(* Logix 5000 project; controller Sucrose_Main Emulate 5570 rev 20.12; software revision 20.01; part 13 of 30 *)
(* tags used below, declared in another part *)
   AI_E21_0 : REAL[8];   // Analog Input EN2T_FLX 192.168.1.21
   AI_E21_1 : REAL[8];   // Analog Input EN2T_FLX 192.168.1.21
   AI_E21_2 : REAL[8];   // Analog Input EN2T_FLX 192.168.1.21
   Rung_Comment : BOOL;
   SucroseCIP_RINGMAIN_REMOTE : CIP_REMOTE;
   SucroseFiltration : Area_Program;
(* FiltrationArea_AutoLogic, continued *)

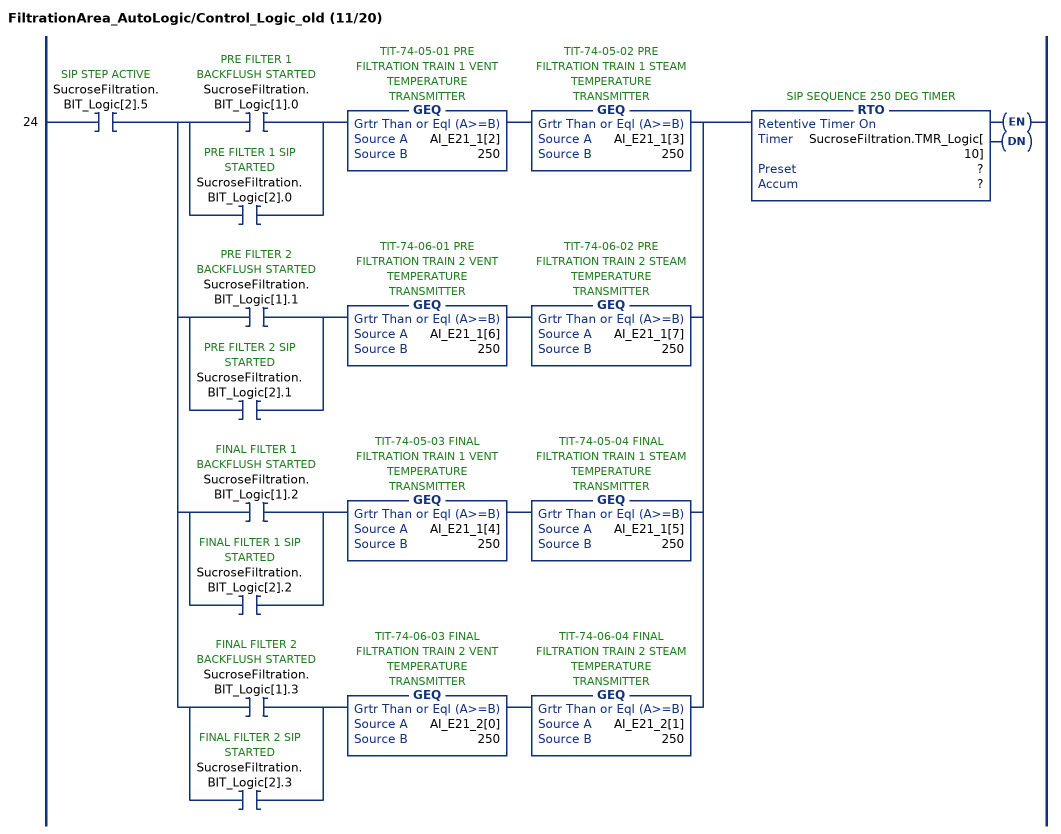
   [picture p232: FiltrationArea_AutoLogic/Control_Logic_old rungs 24-24]
   24: XIC(SucroseFiltration.BIT_Logic[2].5)[[XIC(SucroseFiltration.BIT_Logic[1].0) ,XIC(SucroseFiltration.BIT_Logic[2].0) ] GEQ(AI_E21_1[2],250) GEQ(AI_E21_1[3],250) ,[XIC(SucroseFiltration.BIT_Logic[1].1) ,XIC(SucroseFiltration.BIT_Logic[2].1) ] GEQ(AI_E21_1[6],250) GEQ(AI_E21_1[7],250) ,[XIC(SucroseFiltration.BIT_Logic[1].2) ,XIC(SucroseFiltration.BIT_Logic[2].2) ] GEQ(AI_E21_1[4],250) GEQ(AI_E21_1[5],250) ,[XIC(SucroseFiltration.BIT_Logic[1].3) ,XIC(SucroseFiltration.BIT_Logic[2].3) ] GEQ(AI_E21_2[0],250) GEQ(AI_E21_2[1],250) ]RTO(SucroseFiltration.TMR_Logic[10],?,?);
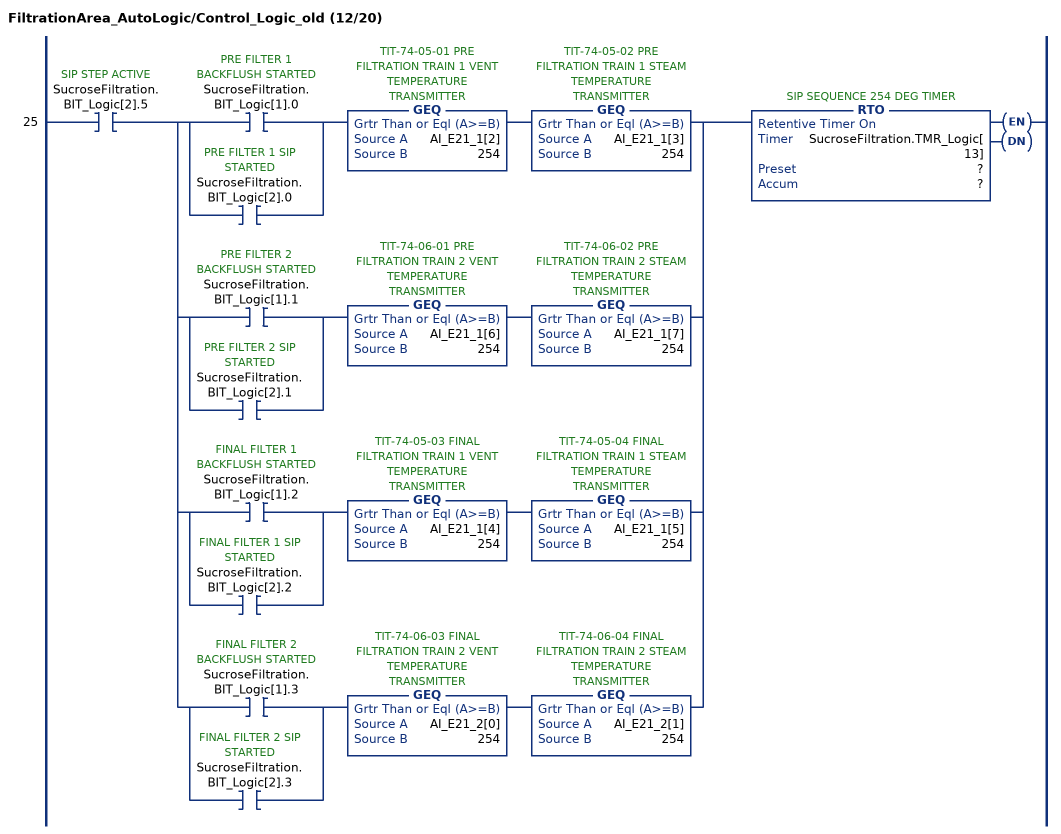
   25: XIC(SucroseFiltration.BIT_Logic[2].5)[[XIC(SucroseFiltration.BIT_Logic[1].0) ,XIC(SucroseFiltration.BIT_Logic[2].0) ] GEQ(AI_E21_1[2],254) GEQ(AI_E21_1[3],254) ,[XIC(SucroseFiltration.BIT_Logic[1].1) ,XIC(SucroseFiltration.BIT_Logic[2].1) ] GEQ(AI_E21_1[6],254) GEQ(AI_E21_1[7],254) ,[XIC(SucroseFiltration.BIT_Logic[1].2) ,XIC(SucroseFiltration.BIT_Logic[2].2) ] GEQ(AI_E21_1[4],254) GEQ(AI_E21_1[5],254) ,[XIC(SucroseFiltration.BIT_Logic[1].3) ,XIC(SucroseFiltration.BIT_Logic[2].3) ] GEQ(AI_E21_2[0],254) GEQ(AI_E21_2[1],254) ]RTO(SucroseFiltration.TMR_Logic[13],?,?);
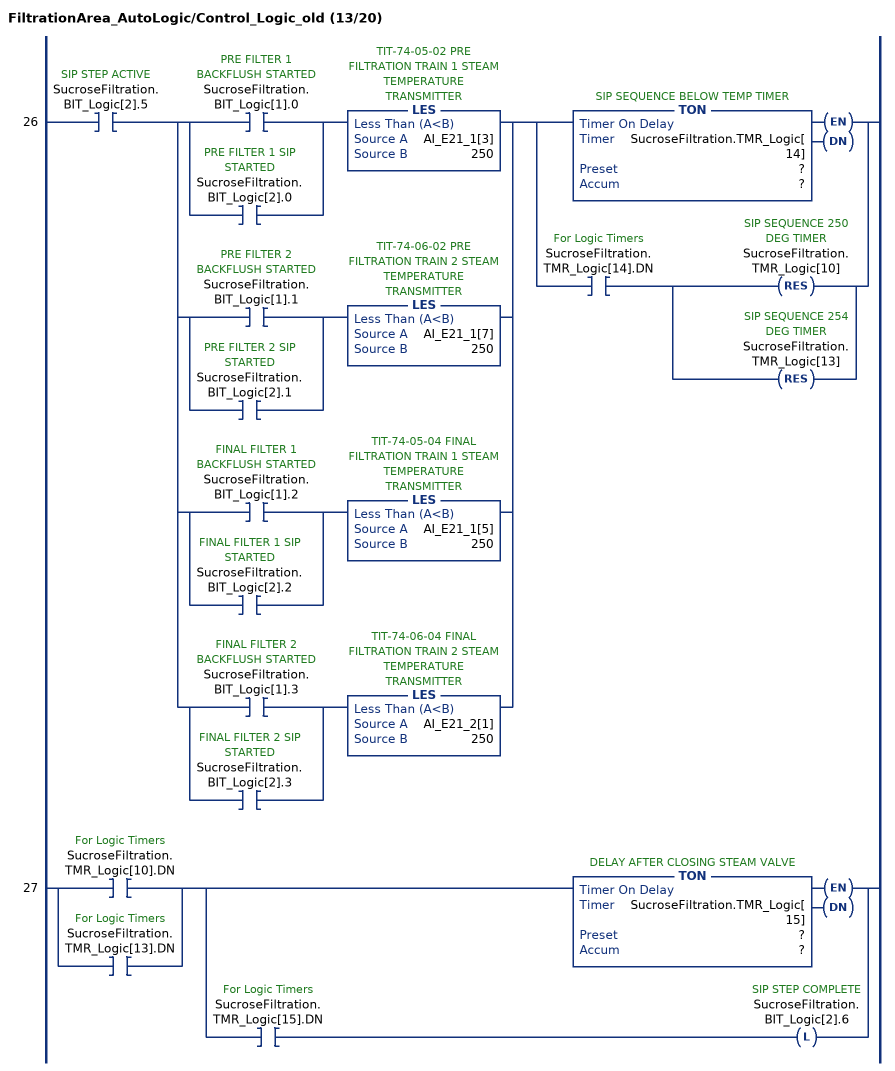
   26: XIC(SucroseFiltration.BIT_Logic[2].5)[[XIC(SucroseFiltration.BIT_Logic[1].0) ,XIC(SucroseFiltration.BIT_Logic[2].0) ] LES(AI_E21_1[3],250) ,[XIC(SucroseFiltration.BIT_Logic[1].1) ,XIC(SucroseFiltration.BIT_Logic[2].1) ] LES(AI_E21_1[7],250) ,[XIC(SucroseFiltration.BIT_Logic[1].2) ,XIC(SucroseFiltration.BIT_Logic[2].2) ] LES(AI_E21_1[5],250) ,[XIC(SucroseFiltration.BIT_Logic[1].3) ,XIC(SucroseFiltration.BIT_Logic[2].3) ] LES(AI_E21_2[1],250) ][TON(SucroseFiltration.TMR_Logic[14],?,?) ,XIC(SucroseFiltration.TMR_Logic[14].DN) [RES(SucroseFiltration.TMR_Logic[10]) ,RES(SucroseFiltration.TMR_Logic[13]) ] ];
   27: [XIC(SucroseFiltration.TMR_Logic[10].DN) ,XIC(SucroseFiltration.TMR_Logic[13].DN) ][TON(SucroseFiltration.TMR_Logic[15],?,?) ,XIC(SucroseFiltration.TMR_Logic[15].DN) OTL(SucroseFiltration.BIT_Logic[2].6) ];
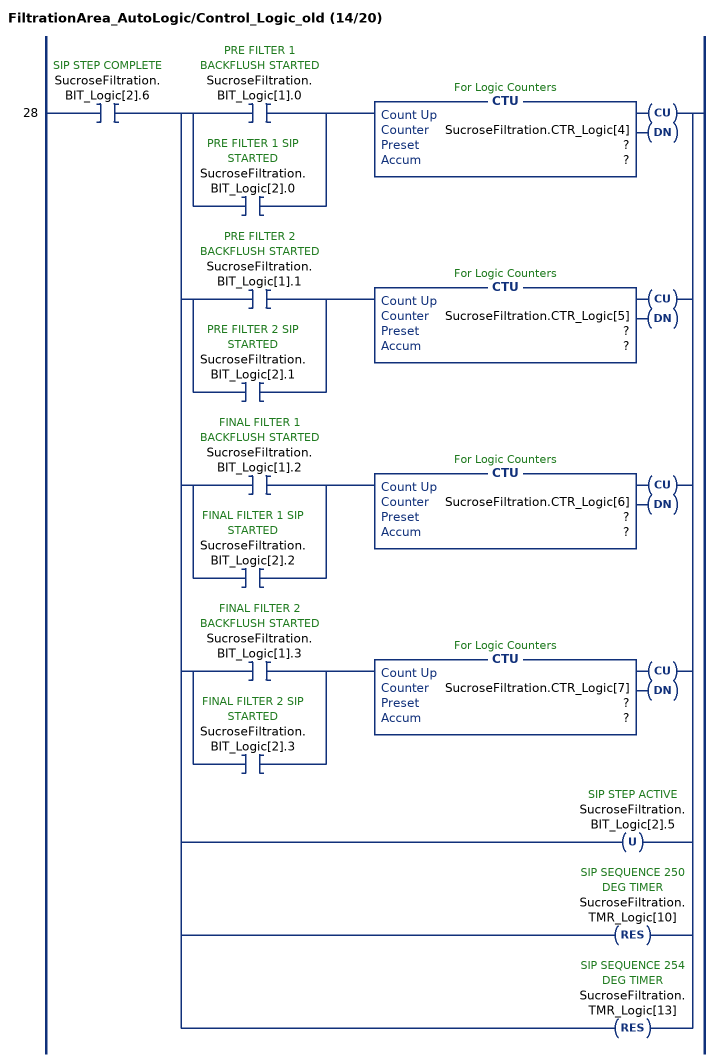
   28: XIC(SucroseFiltration.BIT_Logic[2].6)[[XIC(SucroseFiltration.BIT_Logic[1].0) ,XIC(SucroseFiltration.BIT_Logic[2].0) ] CTU(SucroseFiltration.CTR_Logic[4],?,?) ,[XIC(SucroseFiltration.BIT_Logic[1].1) ,XIC(SucroseFiltration.BIT_Logic[2].1) ] CTU(SucroseFiltration.CTR_Logic[5],?,?) ,[XIC(SucroseFiltration.BIT_Logic[1].2) ,XIC(SucroseFiltration.BIT_Logic[2].2) ] CTU(SucroseFiltration.CTR_Logic[6],?,?) ,[XIC(SucroseFiltration.BIT_Logic[1].3) ,XIC(SucroseFiltration.BIT_Logic[2].3) ] CTU(SucroseFiltration.CTR_Logic[7],?,?) ,OTU(SucroseFiltration.BIT_Logic[2].5) ,RES(SucroseFiltration.TMR_Logic[10]) ,RES(SucroseFiltration.TMR_Logic[13]) ];
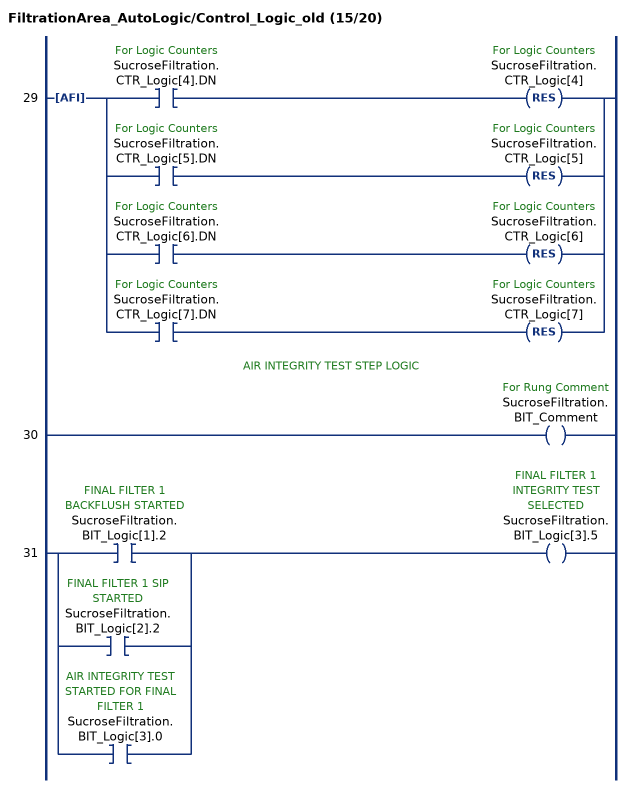
   29: AFI()[XIC(SucroseFiltration.CTR_Logic[4].DN) RES(SucroseFiltration.CTR_Logic[4]) ,XIC(SucroseFiltration.CTR_Logic[5].DN) RES(SucroseFiltration.CTR_Logic[5]) ,XIC(SucroseFiltration.CTR_Logic[6].DN) RES(SucroseFiltration.CTR_Logic[6]) ,XIC(SucroseFiltration.CTR_Logic[7].DN) RES(SucroseFiltration.CTR_Logic[7]) ];
   // AIR INTEGRITY TEST STEP LOGIC
   30: OTE(SucroseFiltration.BIT_Comment);
   31: [XIC(SucroseFiltration.BIT_Logic[1].2) ,XIC(SucroseFiltration.BIT_Logic[2].2) ,XIC(SucroseFiltration.BIT_Logic[3].0) ]OTE(SucroseFiltration.BIT_Logic[3].5);
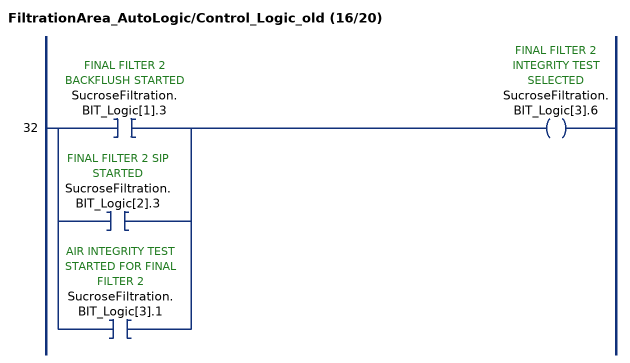
   32: [XIC(SucroseFiltration.BIT_Logic[1].3) ,XIC(SucroseFiltration.BIT_Logic[2].3) ,XIC(SucroseFiltration.BIT_Logic[3].1) ]OTE(SucroseFiltration.BIT_Logic[3].6);
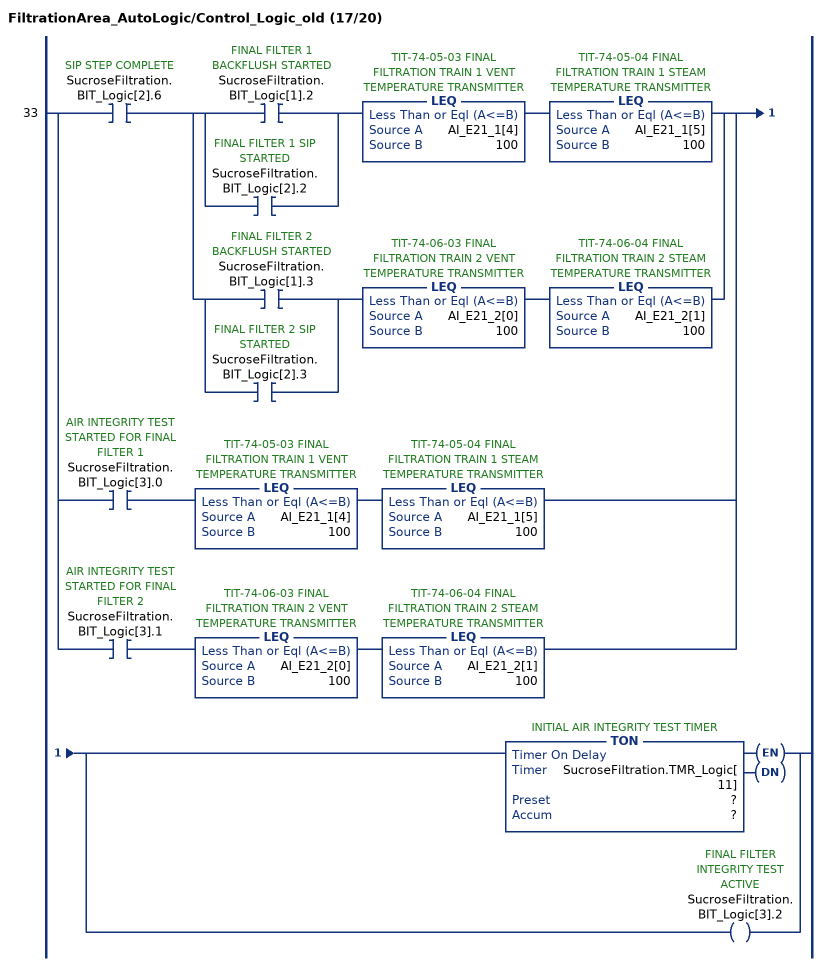
   33: [XIC(SucroseFiltration.BIT_Logic[2].6) [[XIC(SucroseFiltration.BIT_Logic[1].2) ,XIC(SucroseFiltration.BIT_Logic[2].2) ] LEQ(AI_E21_1[4],100) LEQ(AI_E21_1[5],100) ,[XIC(SucroseFiltration.BIT_Logic[1].3) ,XIC(SucroseFiltration.BIT_Logic[2].3) ] LEQ(AI_E21_2[0],100) LEQ(AI_E21_2[1],100) ] ,[XIC(SucroseFiltration.BIT_Logic[3].0) LEQ(AI_E21_1[4],100) LEQ(AI_E21_1[5],100) ,XIC(SucroseFiltration.BIT_Logic[3].1) LEQ(AI_E21_2[0],100) LEQ(AI_E21_2[1],100) ] ][TON(SucroseFiltration.TMR_Logic[11],?,?) ,OTE(SucroseFiltration.BIT_Logic[3].2) ];
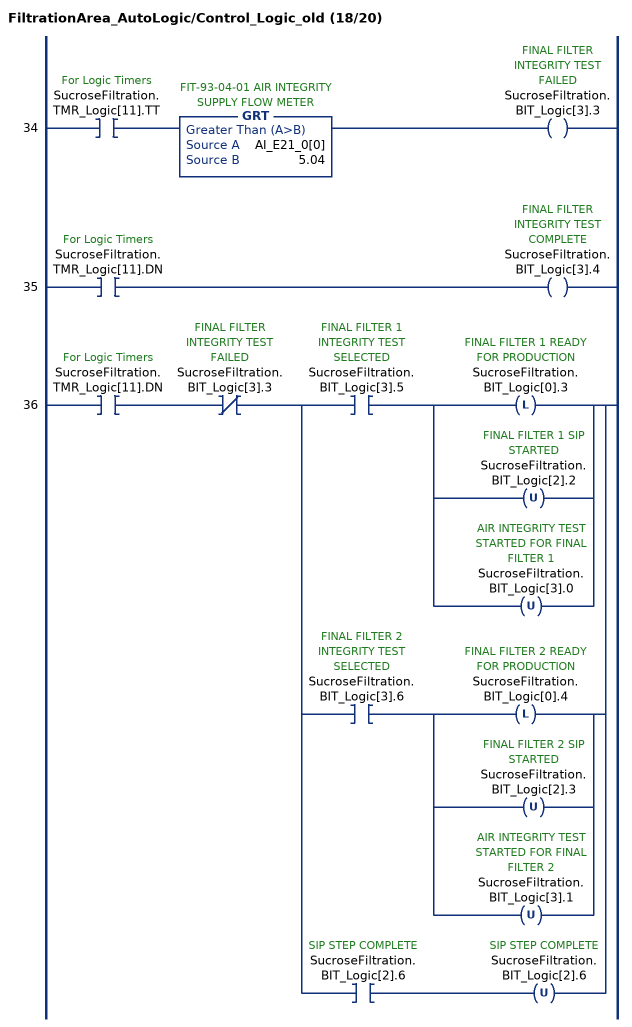
   34: XIC(SucroseFiltration.TMR_Logic[11].TT)GRT(AI_E21_0[0],5.04)OTE(SucroseFiltration.BIT_Logic[3].3);
   35: XIC(SucroseFiltration.TMR_Logic[11].DN)OTE(SucroseFiltration.BIT_Logic[3].4);
   36: XIC(SucroseFiltration.TMR_Logic[11].DN)XIO(SucroseFiltration.BIT_Logic[3].3)[XIC(SucroseFiltration.BIT_Logic[3].5) [OTL(SucroseFiltration.BIT_Logic[0].3) ,OTU(SucroseFiltration.BIT_Logic[2].2) ,OTU(SucroseFiltration.BIT_Logic[3].0) ] ,XIC(SucroseFiltration.BIT_Logic[3].6) [OTL(SucroseFiltration.BIT_Logic[0].4) ,OTU(SucroseFiltration.BIT_Logic[2].3) ,OTU(SucroseFiltration.BIT_Logic[3].1) ] ,XIC(SucroseFiltration.BIT_Logic[2].6) OTU(SucroseFiltration.BIT_Logic[2].6) ];
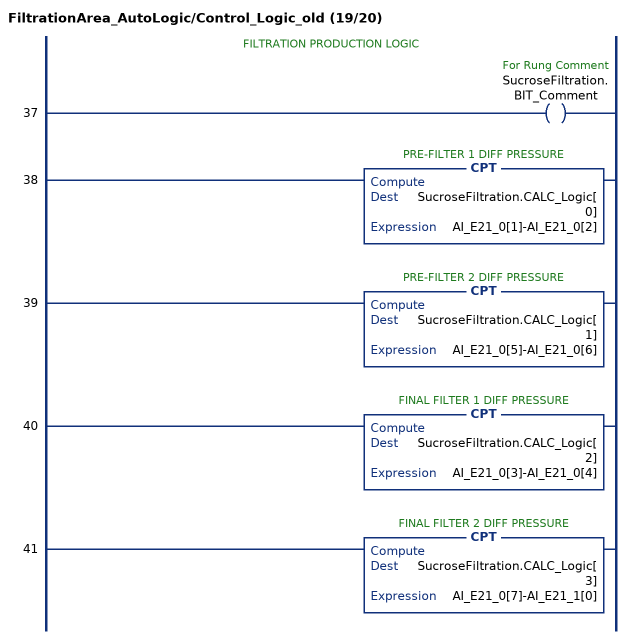
   // FILTRATION PRODUCTION LOGIC
   37: OTE(SucroseFiltration.BIT_Comment);
   38: CPT(SucroseFiltration.CALC_Logic[0],AI_E21_0[1]-AI_E21_0[2]);
   39: CPT(SucroseFiltration.CALC_Logic[1],AI_E21_0[5]-AI_E21_0[6]);
   40: CPT(SucroseFiltration.CALC_Logic[2],AI_E21_0[3]-AI_E21_0[4]);
   41: CPT(SucroseFiltration.CALC_Logic[3],AI_E21_0[7]-AI_E21_1[0]);
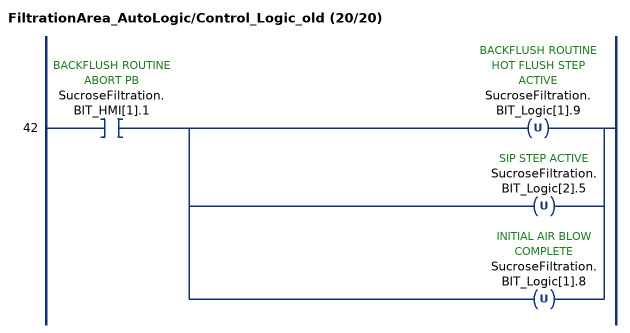
   42: XIC(SucroseFiltration.BIT_HMI[1].1)[OTU(SucroseFiltration.BIT_Logic[1].9) ,OTU(SucroseFiltration.BIT_Logic[2].5) ,OTU(SucroseFiltration.BIT_Logic[1].8) ];
END_ROUTINE

ROUTINE Enable_Logic   (* ladder *)
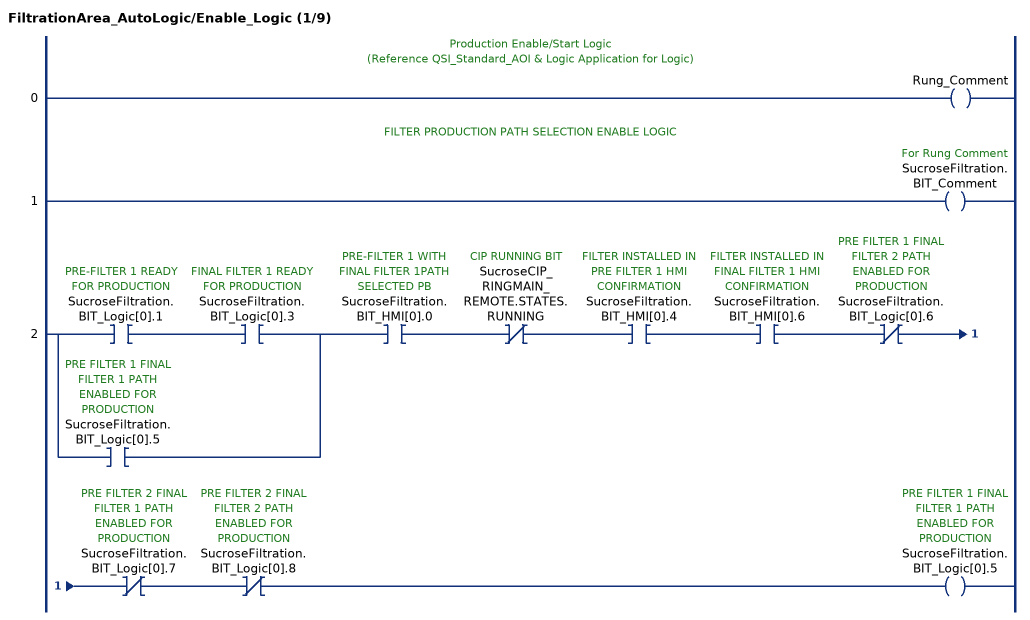
   // Production Enable/Start Logic
   // (Reference QSI_Standard_AOI & Logic Application for Logic)
   0: OTE(Rung_Comment);
   // FILTER PRODUCTION PATH SELECTION ENABLE LOGIC
   1: OTE(SucroseFiltration.BIT_Comment);
   2: [XIC(SucroseFiltration.BIT_Logic[0].1) XIC(SucroseFiltration.BIT_Logic[0].3) ,XIC(SucroseFiltration.BIT_Logic[0].5) ]XIC(SucroseFiltration.BIT_HMI[0].0)XIO(SucroseCIP_RINGMAIN_REMOTE.STATES.RUNNING)XIC(SucroseFiltration.BIT_HMI[0].4)XIC(SucroseFiltration.BIT_HMI[0].6)XIO(SucroseFiltration.BIT_Logic[0].6)XIO(SucroseFiltration.BIT_Logic[0].7)XIO(SucroseFiltration.BIT_Logic[0].8)OTE(SucroseFiltration.BIT_Logic[0].5);
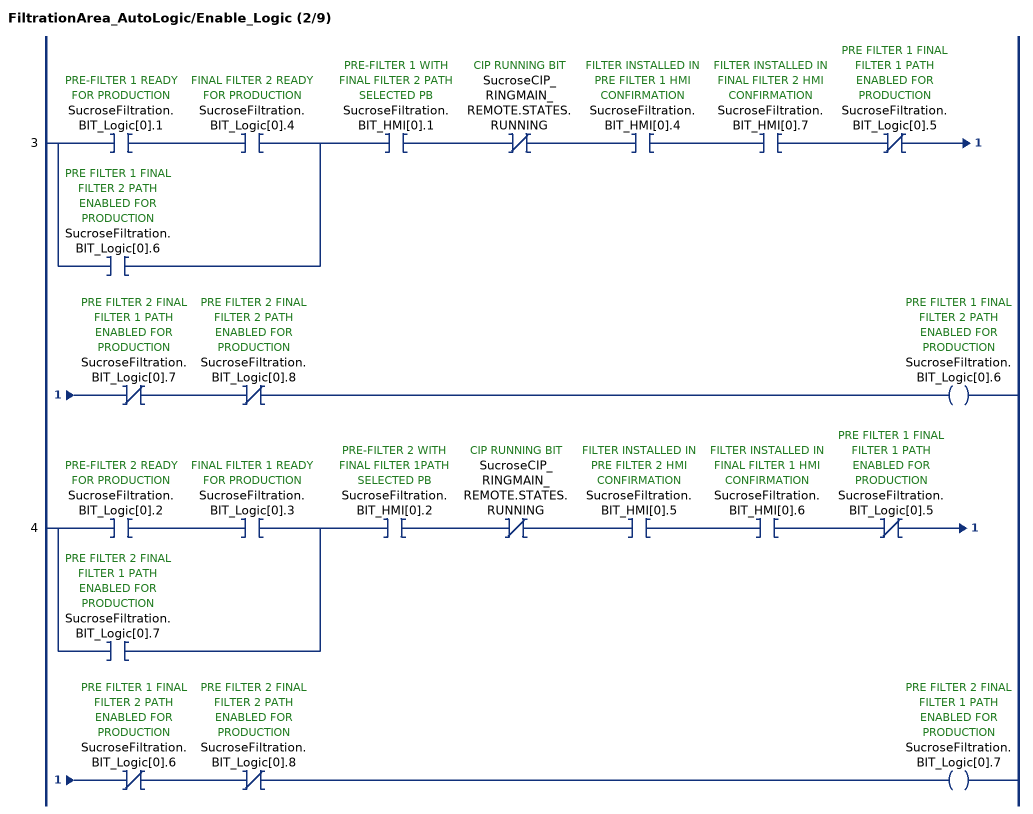
   3: [XIC(SucroseFiltration.BIT_Logic[0].1) XIC(SucroseFiltration.BIT_Logic[0].4) ,XIC(SucroseFiltration.BIT_Logic[0].6) ]XIC(SucroseFiltration.BIT_HMI[0].1)XIO(SucroseCIP_RINGMAIN_REMOTE.STATES.RUNNING)XIC(SucroseFiltration.BIT_HMI[0].4)XIC(SucroseFiltration.BIT_HMI[0].7)XIO(SucroseFiltration.BIT_Logic[0].5)XIO(SucroseFiltration.BIT_Logic[0].7)XIO(SucroseFiltration.BIT_Logic[0].8)OTE(SucroseFiltration.BIT_Logic[0].6);
   4: [XIC(SucroseFiltration.BIT_Logic[0].2) XIC(SucroseFiltration.BIT_Logic[0].3) ,XIC(SucroseFiltration.BIT_Logic[0].7) ]XIC(SucroseFiltration.BIT_HMI[0].2)XIO(SucroseCIP_RINGMAIN_REMOTE.STATES.RUNNING)XIC(SucroseFiltration.BIT_HMI[0].5)XIC(SucroseFiltration.BIT_HMI[0].6)XIO(SucroseFiltration.BIT_Logic[0].5)XIO(SucroseFiltration.BIT_Logic[0].6)XIO(SucroseFiltration.BIT_Logic[0].8)OTE(SucroseFiltration.BIT_Logic[0].7);
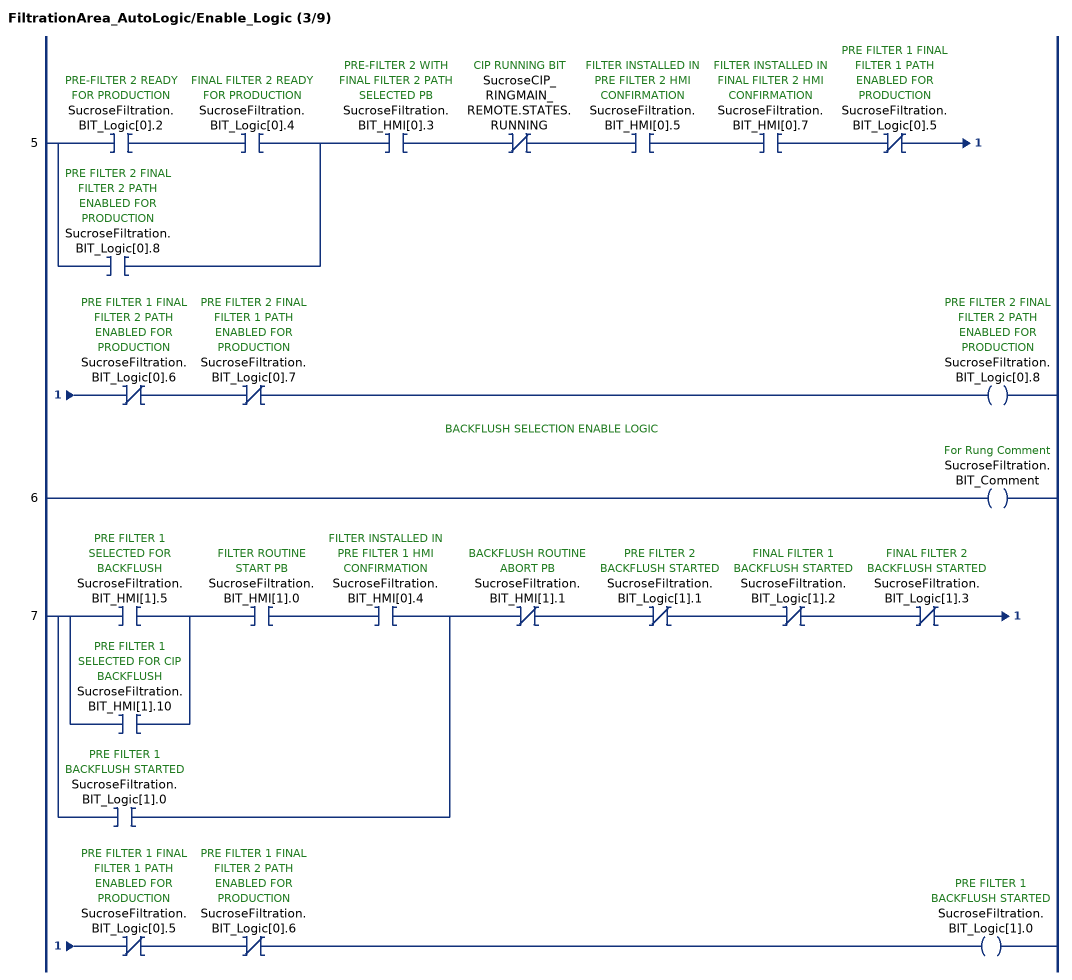
   5: [XIC(SucroseFiltration.BIT_Logic[0].2) XIC(SucroseFiltration.BIT_Logic[0].4) ,XIC(SucroseFiltration.BIT_Logic[0].8) ]XIC(SucroseFiltration.BIT_HMI[0].3)XIO(SucroseCIP_RINGMAIN_REMOTE.STATES.RUNNING)XIC(SucroseFiltration.BIT_HMI[0].5)XIC(SucroseFiltration.BIT_HMI[0].7)XIO(SucroseFiltration.BIT_Logic[0].5)XIO(SucroseFiltration.BIT_Logic[0].6)XIO(SucroseFiltration.BIT_Logic[0].7)OTE(SucroseFiltration.BIT_Logic[0].8);
   // BACKFLUSH SELECTION ENABLE LOGIC
   6: OTE(SucroseFiltration.BIT_Comment);
   7: [[XIC(SucroseFiltration.BIT_HMI[1].5) ,XIC(SucroseFiltration.BIT_HMI[1].10) ] XIC(SucroseFiltration.BIT_HMI[1].0) XIC(SucroseFiltration.BIT_HMI[0].4) ,XIC(SucroseFiltration.BIT_Logic[1].0) ]XIO(SucroseFiltration.BIT_HMI[1].1)XIO(SucroseFiltration.BIT_Logic[1].1)XIO(SucroseFiltration.BIT_Logic[1].2)XIO(SucroseFiltration.BIT_Logic[1].3)XIO(SucroseFiltration.BIT_Logic[0].5)XIO(SucroseFiltration.BIT_Logic[0].6)OTE(SucroseFiltration.BIT_Logic[1].0);
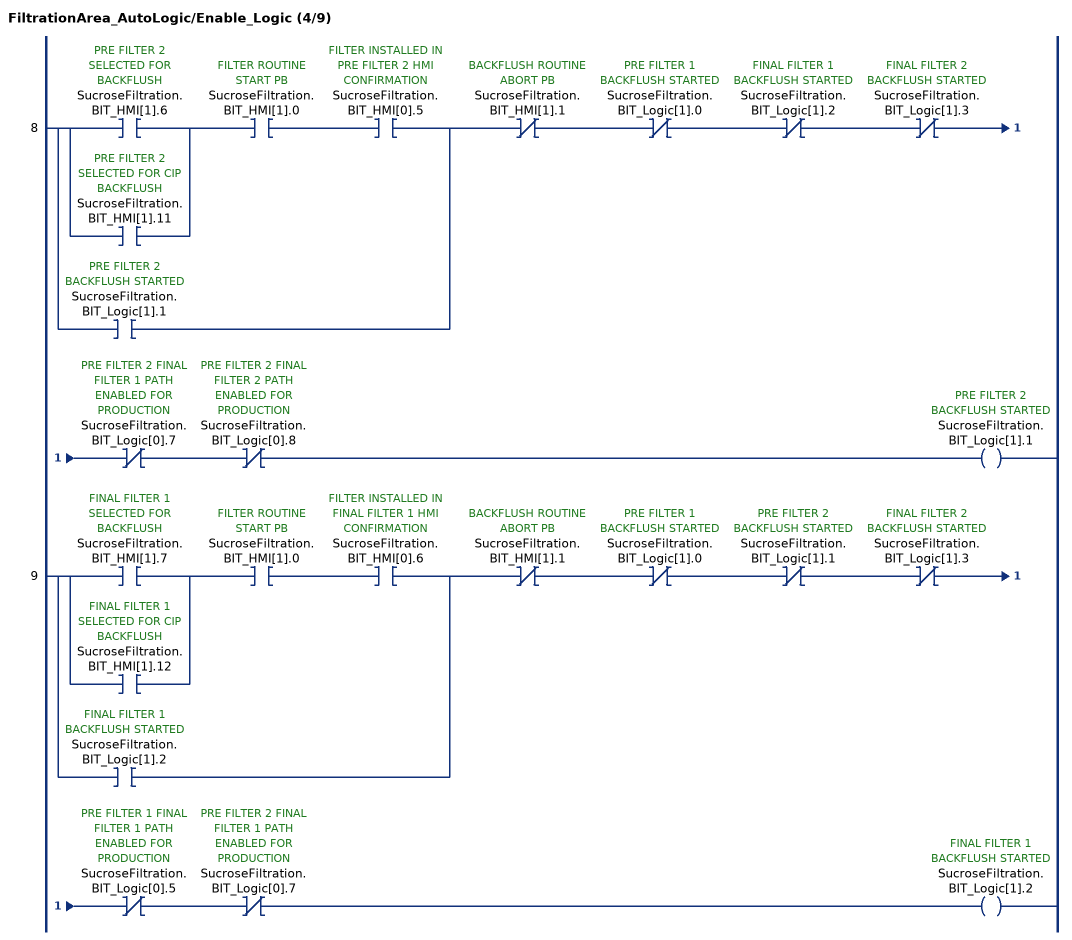
   8: [[XIC(SucroseFiltration.BIT_HMI[1].6) ,XIC(SucroseFiltration.BIT_HMI[1].11) ] XIC(SucroseFiltration.BIT_HMI[1].0) XIC(SucroseFiltration.BIT_HMI[0].5) ,XIC(SucroseFiltration.BIT_Logic[1].1) ]XIO(SucroseFiltration.BIT_HMI[1].1)XIO(SucroseFiltration.BIT_Logic[1].0)XIO(SucroseFiltration.BIT_Logic[1].2)XIO(SucroseFiltration.BIT_Logic[1].3)XIO(SucroseFiltration.BIT_Logic[0].7)XIO(SucroseFiltration.BIT_Logic[0].8)OTE(SucroseFiltration.BIT_Logic[1].1);
   9: [[XIC(SucroseFiltration.BIT_HMI[1].7) ,XIC(SucroseFiltration.BIT_HMI[1].12) ] XIC(SucroseFiltration.BIT_HMI[1].0) XIC(SucroseFiltration.BIT_HMI[0].6) ,XIC(SucroseFiltration.BIT_Logic[1].2) ]XIO(SucroseFiltration.BIT_HMI[1].1)XIO(SucroseFiltration.BIT_Logic[1].0)XIO(SucroseFiltration.BIT_Logic[1].1)XIO(SucroseFiltration.BIT_Logic[1].3)XIO(SucroseFiltration.BIT_Logic[0].5)XIO(SucroseFiltration.BIT_Logic[0].7)OTE(SucroseFiltration.BIT_Logic[1].2);
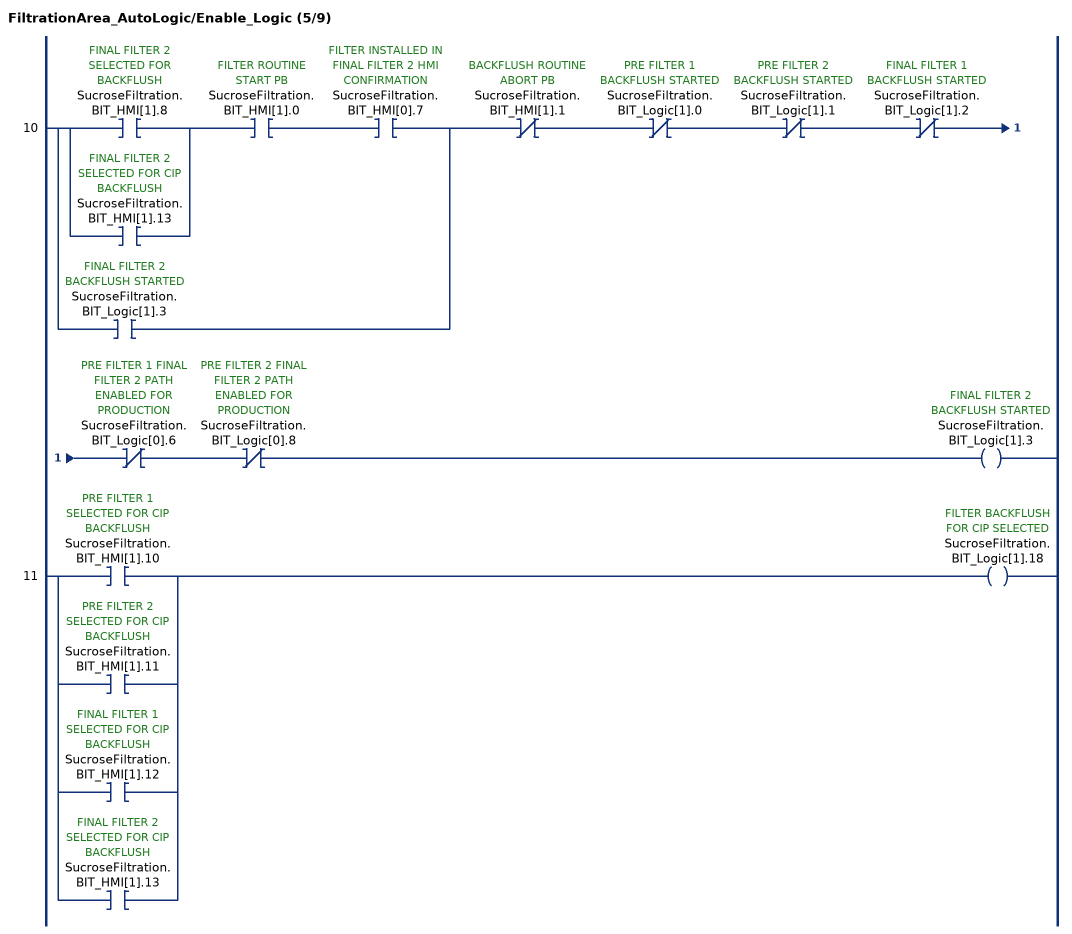
   10: [[XIC(SucroseFiltration.BIT_HMI[1].8) ,XIC(SucroseFiltration.BIT_HMI[1].13) ] XIC(SucroseFiltration.BIT_HMI[1].0) XIC(SucroseFiltration.BIT_HMI[0].7) ,XIC(SucroseFiltration.BIT_Logic[1].3) ]XIO(SucroseFiltration.BIT_HMI[1].1)XIO(SucroseFiltration.BIT_Logic[1].0)XIO(SucroseFiltration.BIT_Logic[1].1)XIO(SucroseFiltration.BIT_Logic[1].2)XIO(SucroseFiltration.BIT_Logic[0].6)XIO(SucroseFiltration.BIT_Logic[0].8)OTE(SucroseFiltration.BIT_Logic[1].3);
   11: [XIC(SucroseFiltration.BIT_HMI[1].10) ,XIC(SucroseFiltration.BIT_HMI[1].11) ,XIC(SucroseFiltration.BIT_HMI[1].12) ,XIC(SucroseFiltration.BIT_HMI[1].13) ]OTE(SucroseFiltration.BIT_Logic[1].18);
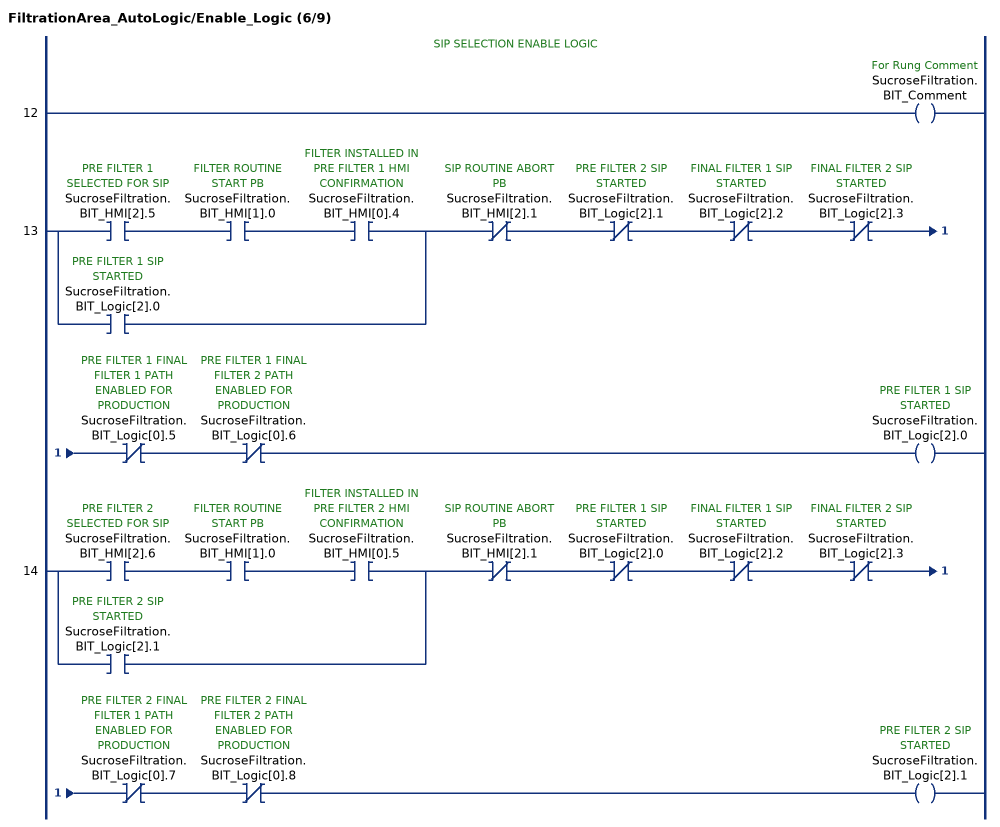
   // SIP SELECTION ENABLE LOGIC
   12: OTE(SucroseFiltration.BIT_Comment);
   13: [XIC(SucroseFiltration.BIT_HMI[2].5) XIC(SucroseFiltration.BIT_HMI[1].0) XIC(SucroseFiltration.BIT_HMI[0].4) ,XIC(SucroseFiltration.BIT_Logic[2].0) ]XIO(SucroseFiltration.BIT_HMI[2].1)XIO(SucroseFiltration.BIT_Logic[2].1)XIO(SucroseFiltration.BIT_Logic[2].2)XIO(SucroseFiltration.BIT_Logic[2].3)XIO(SucroseFiltration.BIT_Logic[0].5)XIO(SucroseFiltration.BIT_Logic[0].6)OTE(SucroseFiltration.BIT_Logic[2].0);
   14: [XIC(SucroseFiltration.BIT_HMI[2].6) XIC(SucroseFiltration.BIT_HMI[1].0) XIC(SucroseFiltration.BIT_HMI[0].5) ,XIC(SucroseFiltration.BIT_Logic[2].1) ]XIO(SucroseFiltration.BIT_HMI[2].1)XIO(SucroseFiltration.BIT_Logic[2].0)XIO(SucroseFiltration.BIT_Logic[2].2)XIO(SucroseFiltration.BIT_Logic[2].3)XIO(SucroseFiltration.BIT_Logic[0].7)XIO(SucroseFiltration.BIT_Logic[0].8)OTE(SucroseFiltration.BIT_Logic[2].1);
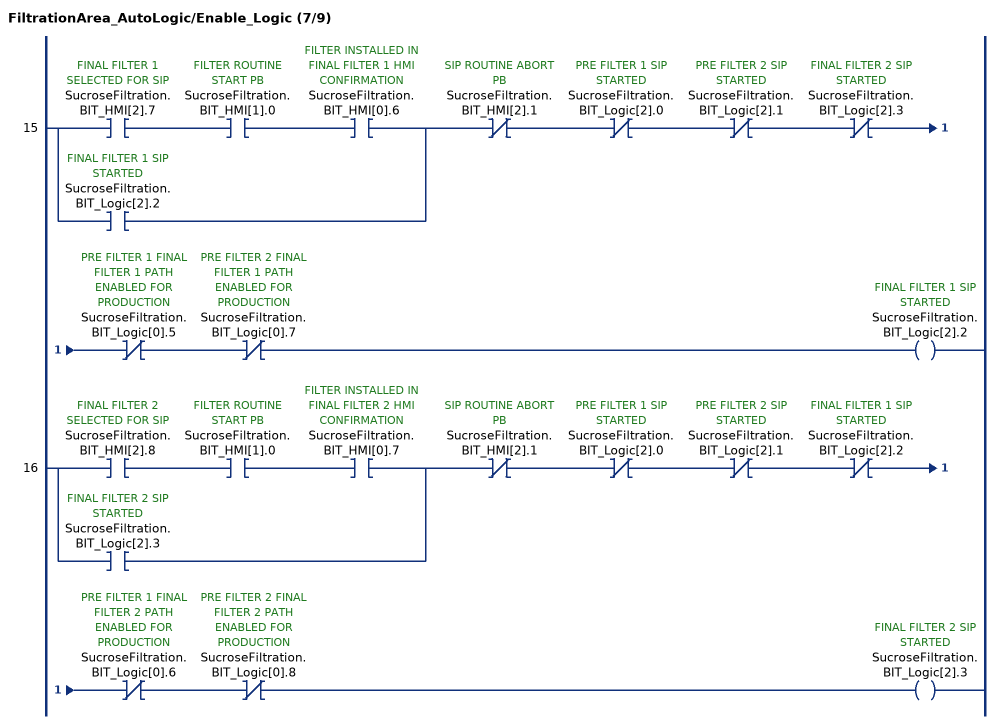
   15: [XIC(SucroseFiltration.BIT_HMI[2].7) XIC(SucroseFiltration.BIT_HMI[1].0) XIC(SucroseFiltration.BIT_HMI[0].6) ,XIC(SucroseFiltration.BIT_Logic[2].2) ]XIO(SucroseFiltration.BIT_HMI[2].1)XIO(SucroseFiltration.BIT_Logic[2].0)XIO(SucroseFiltration.BIT_Logic[2].1)XIO(SucroseFiltration.BIT_Logic[2].3)XIO(SucroseFiltration.BIT_Logic[0].5)XIO(SucroseFiltration.BIT_Logic[0].7)OTE(SucroseFiltration.BIT_Logic[2].2);
   16: [XIC(SucroseFiltration.BIT_HMI[2].8) XIC(SucroseFiltration.BIT_HMI[1].0) XIC(SucroseFiltration.BIT_HMI[0].7) ,XIC(SucroseFiltration.BIT_Logic[2].3) ]XIO(SucroseFiltration.BIT_HMI[2].1)XIO(SucroseFiltration.BIT_Logic[2].0)XIO(SucroseFiltration.BIT_Logic[2].1)XIO(SucroseFiltration.BIT_Logic[2].2)XIO(SucroseFiltration.BIT_Logic[0].6)XIO(SucroseFiltration.BIT_Logic[0].8)OTE(SucroseFiltration.BIT_Logic[2].3);
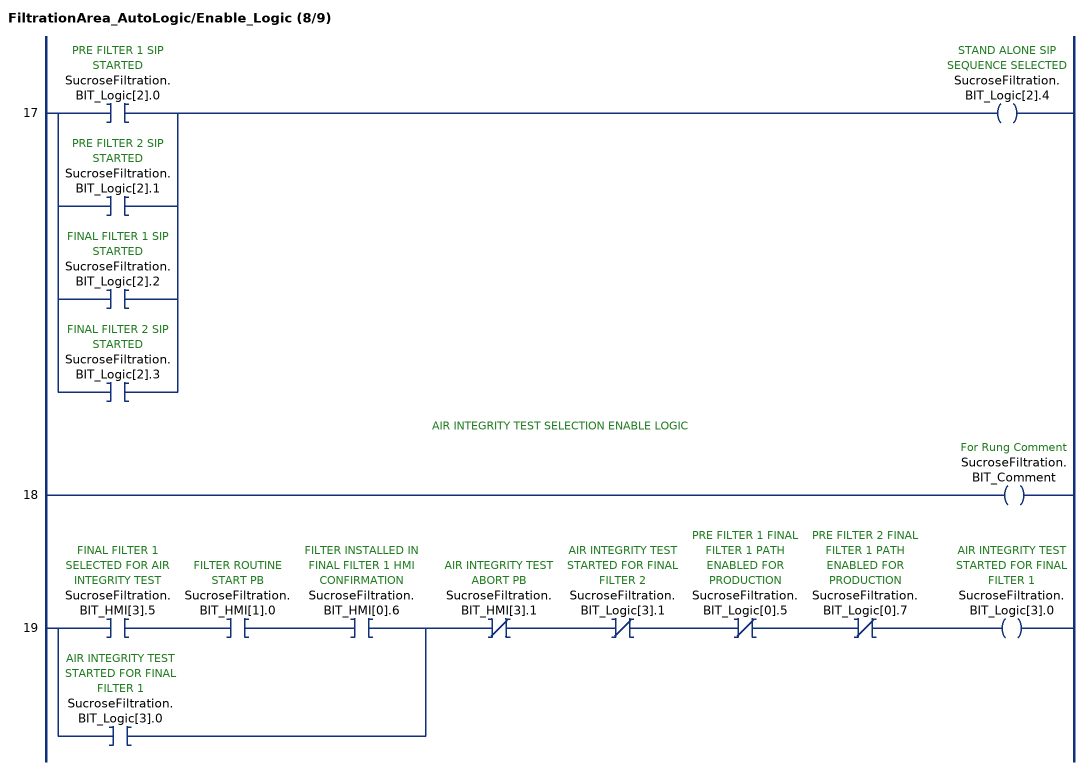
   17: [XIC(SucroseFiltration.BIT_Logic[2].0) ,XIC(SucroseFiltration.BIT_Logic[2].1) ,XIC(SucroseFiltration.BIT_Logic[2].2) ,XIC(SucroseFiltration.BIT_Logic[2].3) ]OTE(SucroseFiltration.BIT_Logic[2].4);
   // AIR INTEGRITY TEST SELECTION ENABLE LOGIC
   18: OTE(SucroseFiltration.BIT_Comment);
   19: [XIC(SucroseFiltration.BIT_HMI[3].5) XIC(SucroseFiltration.BIT_HMI[1].0) XIC(SucroseFiltration.BIT_HMI[0].6) ,XIC(SucroseFiltration.BIT_Logic[3].0) ]XIO(SucroseFiltration.BIT_HMI[3].1)XIO(SucroseFiltration.BIT_Logic[3].1)XIO(SucroseFiltration.BIT_Logic[0].5)XIO(SucroseFiltration.BIT_Logic[0].7)OTE(SucroseFiltration.BIT_Logic[3].0);
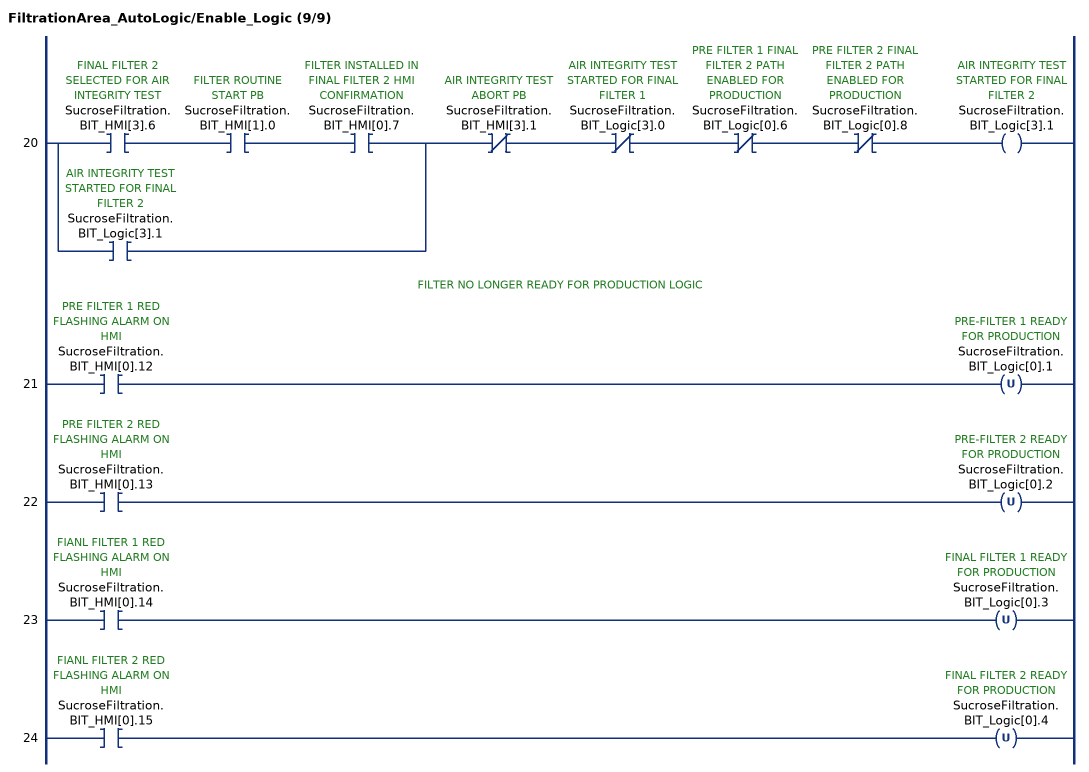
   20: [XIC(SucroseFiltration.BIT_HMI[3].6) XIC(SucroseFiltration.BIT_HMI[1].0) XIC(SucroseFiltration.BIT_HMI[0].7) ,XIC(SucroseFiltration.BIT_Logic[3].1) ]XIO(SucroseFiltration.BIT_HMI[3].1)XIO(SucroseFiltration.BIT_Logic[3].0)XIO(SucroseFiltration.BIT_Logic[0].6)XIO(SucroseFiltration.BIT_Logic[0].8)OTE(SucroseFiltration.BIT_Logic[3].1);
   // FILTER NO LONGER READY FOR PRODUCTION LOGIC
   21: XIC(SucroseFiltration.BIT_HMI[0].12)OTU(SucroseFiltration.BIT_Logic[0].1);
   22: XIC(SucroseFiltration.BIT_HMI[0].13)OTU(SucroseFiltration.BIT_Logic[0].2);
   23: XIC(SucroseFiltration.BIT_HMI[0].14)OTU(SucroseFiltration.BIT_Logic[0].3);
   24: XIC(SucroseFiltration.BIT_HMI[0].15)OTU(SucroseFiltration.BIT_Logic[0].4);
END_ROUTINE
